{attribute addProperty BoxType "EP3351-2022-0016"}
{attribute addProperty Id "AIBridge_InputsAT %I*AIBridge_Inputs_EC606E737290AISupply_InputsAT %I*AISupply_Inputs_EC606E737290WcStateAT %I*WcState_98A4DF7520.250InfoDataAT %I*InfoData_BC63D37F80100"}
{attribute addProperty CRC "2907008076"}
{attribute addProperty SizeInBites "226"}
{attribute addProperty SizeInBytes "28.25"}
TYPE EP3351_952A9D23 :
STRUCT
	{attribute addProperty Name "AIBridge_Inputs"}
	AIBridge_Inputs : AIBridge_Inputs_EC606E73;
	{attribute addProperty Name "AISupply_Inputs"}
	AISupply_Inputs : AISupply_Inputs_EC606E73;
	{attribute addProperty Name "WcState"}
	WcState : WcState_98A4DF75;
	{attribute addProperty Name "InfoData"}
	InfoData : InfoData_BC63D37F;
END_STRUCT
END_TYPE

(* stored: Version 1.2.0.0, ProductVersion 3.1.4024.9
   DUT EP3351_952A9D23: Id {06bdf91b-9c13-4c5f-998c-948f80134342} *)
